// TIA Portal V20 export
DATA_BLOCK "zPMC_Checksum_DB"   // DB390
// stored: InstanceOfName CITI_Logic.zPMC_Checksum, InstanceOfType FB, Namespace CITI_Logic
"CITI_Logic.zPMC_Checksum"
   // VAR_INPUT
   //    IN_Checksum_2 : DWord;
   //    IN_Checksum_3 : DWord;
   //    IN_Checksum_4 : DWord;
   //    IN_Checksum_5 : DWord;
   //    IN_Checksum_6 : DWord;
   //    IN_Checksum_7 : DWord;
   //    IN_Checksum_8 : DWord;
   //    IN_Checksum_9 : DWord;
   //    IN_Checksum_10 : DWord;
   //    IN_Checksum_11 : DWord;
   //    IN_Checksum_12 : DWord;
   //    IN_Checksum_13 : DWord;
   //    IN_Checksum_14 : DWord;
   //    IN_Checksum_15 : DWord;
   //    IN_Checksum_16 : DWord;
   // END_VAR
   // VAR_OUTPUT
   //    Checksum_Out : Array[1..16] of DWord;
   // END_VAR
   // VAR
   //    ON { ExternalAccessible := 'False'; ExternalVisible := 'False'; ExternalWritable := 'False'} : Bool;
   //    OFF { ExternalAccessible := 'False'; ExternalVisible := 'False'; ExternalWritable := 'False'} : Bool;
   // END_VAR
BEGIN
END_DATA_BLOCK
